// TIA Portal V19 export
DATA_BLOCK "A04_DEBUG"   // DB213
// stored: MemoryReserve 100
   VAR
      Force_Sinamics_Infeed_ON : Bool;
      Force_Sinamics_Drives_CtrlSafe : Bool;
      Forse_Contactors_CtrlSafe : Bool;
      LsStratoDepositato : Bool;
      CIn_Manager_DEBUG : Struct
         PareggiatoreTesta : Struct
            Ax : "Positioning_EPOS_Machine_COut";
         END_STRUCT;
         PareggiatoreCoda : Struct
            Ax : "Positioning_EPOS_Machine_COut";
         END_STRUCT;
         Spalle : Struct
            Testa : Struct
               Ax : "Positioning_DOL_Machine_COut";
            END_STRUCT;
            Coda : Struct
               Ax : "Positioning_DOL_Machine_COut";
            END_STRUCT;
         END_STRUCT;
         Spintore : Struct
            Vrt : "ValveMachine_COut";
            Orz : "ValveMachine_COut";
         END_STRUCT;
         TraslazioneStrato : Struct
            Ax_Testa : "Positioning_EPOS_Machine_COut";
            Ax_Coda : "Positioning_EPOS_Machine_COut";
            Manip_Sostegno : "ValveMachine_COut";
            Manip_Pareggiatore : "ValveMachine_COut";
            SostegnoVrt : "ValveMachine_COut";
         END_STRUCT;
         Sollevamento : Struct
            Ax_Testa : "Positioning_DOL_Machine_COut";
            Ax_Coda : "Positioning_DOL_Machine_COut";
         END_STRUCT;
         Sostegno : Struct
            Testa : Struct
               Ax : "Positioning_DOL_Machine_COut";
               Paletto : Struct
                  CtrlSafe : Bool;
                  Standstill : Bool;
                  Rest_CheckNext : Bool;
                  Work_CheckNext : Bool;
                  Pos : Int;
                  RestPosition : Bool;
               END_STRUCT;
            END_STRUCT;
            Coda : Struct
               Ax : "Positioning_DOL_Machine_COut";
               Paletto : Struct
                  CtrlSafe : Bool;
                  Standstill : Bool;
                  Rest_CheckNext : Bool;
                  Work_CheckNext : Bool;
                  Pos : Int;
                  RestPosition : Bool;
               END_STRUCT;
            END_STRUCT;
         END_STRUCT;
         Navetta : Struct
            ReadyToRecive : Bool;
            OutOfWorkspace : Bool;
            InPosizioneDiDeposito : Bool;
            RequestDeposito : Bool;
         END_STRUCT;
      END_STRUCT;
      CIn_Manager04_Debug : Struct
         Navetta : Struct
            Testa : Struct
               Ax : "Positioning_DOL_Machine_COut";
               PalettiEsterni : "ValveMachine_COut";
               PalettiInterni : "ValveMachine_COut";
            END_STRUCT;
            Coda : Struct
               Ax : "Positioning_DOL_Machine_COut";
               PalettiEsterni : "ValveMachine_COut";
               PalettiInterni : "ValveMachine_COut";
            END_STRUCT;
            Cumulativo : Struct
               PalettiEsterni : "ValveMachine_COut";
               PalettiInterni : "ValveMachine_COut";
            END_STRUCT;
         END_STRUCT;
         Sollevamento : Struct
            ReadyToDrop : Bool;   // In posizione di deposito e pacco completato
         END_STRUCT;
         Antiribaltamento : Struct
            Work : Bool;
            Rest : Bool;
         END_STRUCT;
      END_STRUCT;
      Beams_Data : "Prod_Beam_Data";
      O_ID { S7_SetPoint := 'True'} : Int;
   END_VAR
BEGIN
   Beams_Data.O_ACT.O_ID := 2;
   Beams_Data.O_ACT.PPrf_No := 107;
   Beams_Data.O_ACT.MES_IDP := 'HMI';
   Beams_Data.O_ACT.MES_PPrf_Name := 'S120x45x1.25';
   Beams_Data.O_ACT.Beam_Code := 1;
   Beams_Data.O_ACT.Beams_W_A := 45.0;
   Beams_Data.O_ACT.Beams_H_B := 120.0;
   Beams_Data.O_ACT.Beams_Thickness := 1.25;
   Beams_Data.O_ACT.Beams_Len_Min := 999.0;
   Beams_Data.O_ACT.Beams_Len_Max := 1000.0;
   Beams_Data.O_ACT.Beams_Len := 1820.0;
   Beams_Data.O_ACT.Parts_Len := 1820.0;
   Beams_Data.O_ACT.Parts_Tol := 0.0;
   Beams_Data.O_ACT.PackLayout_BeamsPerLayer := 5;
   Beams_Data.O_ACT.PackLayout_Layers_Qty := 5;
END_DATA_BLOCK
